FUNCTION_BLOCK MakeNewRecipe
VAR_IN_OUT
	NumberOfMovements: INT;
	MovementList: ARRAY[1..NumberOfMovements] OF INT;
	MovementMotors: ARRAY[1..NumberOfMovements] OF Motor;
END_VAR
VAR_OUTPUT
	NewRecipe: Recipe;
END_VAR
VAR
END_VAR

IF Automatic.RecipesIndex <= Automatic.MaxNumberOfRecipes THEN
	NewRecipe.NoOfMovements := NumberOfMovements;
	NewRecipe.MovementList := MovementList;
	NewRecipe.MovementMotors := MovementMotors;
	
	Automatic.Recipes[Automatic.RecipesIndex] := NewRecipe;
	Automatic.RecipesIndex := Automatic.RecipesIndex + 1;
END_IF

END_FUNCTION_BLOCK

(* stored: Version 1.1.0.1, ProductVersion 3.1.4024.13
   POU MakeNewRecipe: Id {46a50fc8-6651-4bb7-bd5b-aa4aa95e59d3}, SpecialFunc None *)
